(* IEC 61131-3 sources: YaoKangDeviceDemo/src/20_Decision, 3 files *)

(* ---- PRG_ErrorManager.st ---- *)
(*============================================================================
  PRG_ErrorManager —— 层 20 决策：错误与诊断（扫描链第 4 环），错误唯一写入者
  ----------------------------------------------------------------------------
  唯一写入：HMI.Sys.Error（当前活动错误）、HMI.Sys.Warning（警告通道）、
            HMI.Sys.ErrorQueue（9 条环形历史队列）；消费应答 gFaultSubmit:=FALSE。
  读入：  全局故障提交区 gFault*（各任务模块置位 gFaultSubmit 提交，本程序消费）；
          trigAckError / trigSysReset（错误确认/复位脉冲，由 INPUT_ADAPTER 锁存）；
          bSafetyStop（安全链态，活动 Critical 错误在安全链恢复前禁止清除）。
  提交约定：任务模块填 gFaultLevel/Code/Source/SubCode/Val1/Val2 后置
            gFaultSubmit:=TRUE；本程序入队并在同扫描清 gFaultSubmit。
            级别：0=L0 Info 1=L1 Warning 2=L2 Critical。
  清除语义：
    - Critical(L2) 进 Sys.Error 锁存，bNeedReset=TRUE，须 trigAckError/trigSysReset
      且安全链恢复(bSafetyStop=FALSE)才清除；复位不丢历史队列。
    - Warning(L1) 进 Sys.Warning，trigAckError 立即清除，否则存活 10s 自动消退。
    - 队列仅滚动追加，不随复位删除；bOverflow 记录溢出。
  说明：HMI.Sys.Display 的 iErrorCode/iErrorLevel/iErrorSubCode/iErrorSource 由
        HMI_OUTPUT 从 Sys.Error 镜像（单写源：Display 归 HMI_OUTPUT）。
        时间戳为毫秒运行刻度 diMsTick（上电起 ms，MONITOR 每扫累加 SCAN_PERIOD_MS）；
        非日历时钟，日志若需年月日时分秒待现场引入 RTC 库 FB 后替换（见 GVL_Internal diMsTick TODO）。
==========================================================================*)
PROGRAM PRG_ErrorManager

(*------------------------------------------------------------
  1) 故障消费：入队 + 活动错误/警告通道
------------------------------------------------------------*)
IF gFaultSubmit THEN
    (*--- 入环形队列：9 条，iTail 推进、iCount 计数、溢出置位 ---*)
    HMI.Sys.ErrorQueue.aEntries[HMI.Sys.ErrorQueue.iTail].iLevel      := gFaultLevel;
    HMI.Sys.ErrorQueue.aEntries[HMI.Sys.ErrorQueue.iTail].iCode       := gFaultCode;
    HMI.Sys.ErrorQueue.aEntries[HMI.Sys.ErrorQueue.iTail].iSource     := gFaultSource;
    HMI.Sys.ErrorQueue.aEntries[HMI.Sys.ErrorQueue.iTail].iVal1       := gFaultVal1;
    HMI.Sys.ErrorQueue.aEntries[HMI.Sys.ErrorQueue.iTail].diTimestamp := diMsTick;  (* 事件毫秒刻度（上电起 ms）；日历 RTC 待现场引入库 FB，见 GVL_Internal diMsTick TODO *)

    HMI.Sys.ErrorQueue.iTail := HMI.Sys.ErrorQueue.iTail + 1;
    IF HMI.Sys.ErrorQueue.iTail >= 9 THEN
        HMI.Sys.ErrorQueue.iTail := 0;
    END_IF;

    IF HMI.Sys.ErrorQueue.iCount < 9 THEN
        HMI.Sys.ErrorQueue.iCount := HMI.Sys.ErrorQueue.iCount + 1;
    ELSE
        HMI.Sys.ErrorQueue.iHead := HMI.Sys.ErrorQueue.iHead + 1;  (* 滚动覆盖最旧 *)
        IF HMI.Sys.ErrorQueue.iHead >= 9 THEN
            HMI.Sys.ErrorQueue.iHead := 0;
        END_IF;
        HMI.Sys.ErrorQueue.bOverflow := TRUE;
    END_IF;

    (*--- 当前活动错误 / 警告通道（L2→Error 锁存，L1→Warning 通道，L0 仅入队） ---*)
    IF gFaultLevel >= 2 THEN
        HMI.Sys.Error.iLevel     := gFaultLevel;
        HMI.Sys.Error.iCode      := gFaultCode;
        HMI.Sys.Error.iSource    := gFaultSource;
        HMI.Sys.Error.iSubCode   := gFaultSubCode;
        HMI.Sys.Error.iVal1      := gFaultVal1;
        HMI.Sys.Error.iVal2      := gFaultVal2;
        HMI.Sys.Error.bActive    := TRUE;
        HMI.Sys.Error.bCritical  := TRUE;
        HMI.Sys.Error.bEscalated := (gFaultCode = ERR_SOFT_ESTOP_TOUT);  (* 软急停超时升级硬急停 *)
        HMI.Sys.Error.bNeedReset := TRUE;    (* Critical 一律需手动复位 *)
    ELSIF gFaultLevel = 1 THEN
        HMI.Sys.Warning.iCode   := gFaultCode;
        HMI.Sys.Warning.iSource := gFaultSource;
        HMI.Sys.Warning.iVal1   := gFaultVal1;
        HMI.Sys.Warning.bActive := TRUE;
    END_IF;

    gFaultSubmit := FALSE;   (* 消费应答 *)
END_IF;

(*------------------------------------------------------------
  2) 活动 Critical 错误清除：确认/复位脉冲 + 安全链已恢复
     （安全链未恢复时拒绝清除，防止带故障复位运行）
------------------------------------------------------------*)
IF HMI.Sys.Error.bActive AND HMI.Sys.Error.bNeedReset THEN
    IF (trigAckError OR trigSysReset) AND NOT bSafetyStop THEN
        HMI.Sys.Error.bActive    := FALSE;
        HMI.Sys.Error.bCritical  := FALSE;
        HMI.Sys.Error.bEscalated := FALSE;
        HMI.Sys.Error.bNeedReset := FALSE;
        HMI.Sys.Error.iLevel     := 0;
        HMI.Sys.Error.iCode      := 0;
        HMI.Sys.Error.iSource    := 0;
        HMI.Sys.Error.iSubCode   := 0;
        HMI.Sys.Error.iVal1      := 0;
        HMI.Sys.Error.iVal2      := 0;
    END_IF;
END_IF;

(*------------------------------------------------------------
  3) 警告通道：确认即清；否则存活 10s 自动消退（实时态类警告）
------------------------------------------------------------*)
TONR(IN := HMI.Sys.Warning.bActive, PT := 10000, Q => emTWarnAge);  (* PT=DINT 毫秒：10s=10000ms *)
IF HMI.Sys.Warning.bActive THEN
    IF trigAckError OR emTWarnAge THEN
        HMI.Sys.Warning.bActive := FALSE;
        HMI.Sys.Warning.iCode   := 0;
        HMI.Sys.Warning.iSource := 0;
        HMI.Sys.Warning.iVal1   := 0;
    END_IF;
END_IF;

END_PROGRAM

(* ---- PRG_ModeManager.st ---- *)
(*============================================================================
  PRG_ModeManager —— 层 20 决策：系统状态机（扫描链第 6 环），iState 唯一写入者
  ----------------------------------------------------------------------------
  唯一写入：iState / iWorkMode / iUserRole / iBlockReason（全局）；
            Sys.Status 的 iState/iHealthLevel/diReadyCheckResult/bReady/
            bSafeToStart/bAutoProcessRunning/bIsEmergency/bNeedReset；
            离态残留电平命令（axisJogPos/axisJogNeg/jogPushUp/jogPushDown/pushEnableReq）。
  读入：  安全态 bHardEstop/bSoftEstop/bSafetyStop（最高优先级）；
          trig* 脉冲位（INPUT_ADAPTER 单扫锁存）、HMI.Sys.Cmd 的电平/INT 字段
          （iUserRole/iAuthCode/iWorkMode/bServiceAuthConfirm/bNoLoadConfirm）；
          资格位 bAllAxesIdle/Ref/AtInit、bParamBootDone/bRunParamValid；
          任务上报：Condition.Status.bDone/bError、HMI.Sys.Status.bSelfTestDone。
  规则：任务模块不直接切态，只上报 iPhase 与任务状态位；切换须过门控
        （角色/权限码/资格/安全），门控拒绝写 iBlockReason（45xx）供 HMI 提示；
        急停态无条件穿透；离态清残留电平命令。
  READY_CHECK：diReadyCheckResult 为位掩码（READY_MASK_*），0=全过；不齐时
        每 100 扫提交一次 7001 Warning，掩码值随 iVal1 上报。
==========================================================================*)
PROGRAM PRG_ModeManager

(*============================================================================
  0. 每扫公共计算：角色/工作模式镜像 + 六项资格掩码 + 汇总状态
  ==========================================================================*)
(*--- 工程师双重门控：角色 + 权限码 16#5A ---*)
mmBEngineer := (HMI.Sys.Cmd.iUserRole = ROLE_ENGINEER)
         AND (HMI.Sys.Cmd.iAuthCode = AUTH_CODE_ENGINEER);
iUserRole := HMI.Sys.Cmd.iUserRole;   (* 角色镜像（操作员/工程师） *)

(*--- 六项资格掩码（位值见 GVL_CONST READY_MASK_*，预计算位值直接 OR；LiteST 的 SHL/SHR 第一操作数不能是常量） ---*)
mmDiMask := 0;
IF NOT bAllAxesRef THEN
    mmDiMask := mmDiMask OR READY_MASK_REF;      (* bit5 参考无效 *)
END_IF;
IF NOT bRunParamValid OR NOT bParamBootDone THEN
    mmDiMask := mmDiMask OR READY_MASK_PARAM;   (* bit1 参数无效 *)
END_IF;
IF NOT HMI.Sys.Status.bPowerOn THEN
    mmDiMask := mmDiMask OR READY_MASK_HW;      (* bit2 硬件未上电 *)
END_IF;
IF HMI.Sys.Error.bActive THEN
    mmDiMask := mmDiMask OR READY_MASK_HEALTH;  (* bit3 活动 Critical *)
END_IF;
IF NOT bAllAxesAtInit THEN
    mmDiMask := mmDiMask OR READY_MASK_POS;     (* bit4 未在初始位 *)
END_IF;
IF NOT (retainZeroComm[0] AND retainZeroComm[1] AND retainZeroComm[2] AND retainTailZeroComm) THEN
    mmDiMask := mmDiMask OR READY_MASK_ZERO;    (* bit0 未建零 *)
END_IF;
mmBReadyAll := (mmDiMask = 0);

(*--- 汇总状态回填 Sys.Status ---*)
HMI.Sys.Status.iState             := iState;
HMI.Sys.Status.diReadyCheckResult := mmDiMask;
HMI.Sys.Status.bReady             := (iState = ST_STANDBY) AND mmBReadyAll;
HMI.Sys.Status.bSafeToStart       := mmBReadyAll AND (iState = ST_STANDBY)
                                AND NOT bSafetyStop AND NOT bHardEstop AND NOT bSoftEstop;
HMI.Sys.Status.bIsEmergency       := bHardEstop OR bSoftEstop OR bSafetyStop;
HMI.Sys.Status.bNeedReset         := HMI.Sys.Error.bNeedReset OR HMI.Sys.Error.bActive;
HMI.Sys.Status.bAutoProcessRunning:= (iState = ST_AUTORUN);
HMI.Sys.Status.iWorkMode          := iWorkMode;

(*--- 跳过自检资格位（P11） ---*)
(* 操作员快速启动：六项资格齐（含参考/建零），自检可安全省略；任何活动错误撤销资格 *)
HMI.Sys.Status.bSkipSelfTestAllowed := mmBReadyAll AND NOT HMI.Sys.Error.bActive;
(* 工程师强制跳过：需工程师双重门控（角色+权限码 16#5A），不受就绪位限制 *)
HMI.Sys.Status.bForceSkipSelfTestAllowed := mmBEngineer;

(*--- 健康等级 ---*)
IF HMI.Sys.Error.bActive THEN
    HMI.Sys.Status.iHealthLevel := HEALTH_FAULT;      (* 0 故障 *)
ELSIF HMI.Sys.Warning.bActive THEN
    HMI.Sys.Status.iHealthLevel := HEALTH_WARNING;    (* 2 警告 *)
ELSIF mmBReadyAll THEN
    HMI.Sys.Status.iHealthLevel := HEALTH_NORMAL;     (* 1 正常 *)
ELSE
    HMI.Sys.Status.iHealthLevel := HEALTH_UNKNOWN;    (* 3 未就绪 *)
END_IF;

(*--- 阻塞原因 iBlockReason（MODE_MANAGER 唯一写；稳态原因为主，下方 CASE 内
       工程师门控拒绝分支以 4503 覆盖本扫值）。安全/故障优先，其余按就绪缺项；
       0=无阻塞。与 diReadyCheckResult 掩码并行：掩码供调试，原因码供 HMI 显示。 ---*)
iBlockReason := 0;
IF bHardEstop OR bSoftEstop OR bSafetyStop THEN
    iBlockReason := BLOCK_REASON_SAFETY;   (* 4501 安全链动作（急停/保护停机中） *)
ELSIF HMI.Sys.Error.bActive THEN
    iBlockReason := BLOCK_REASON_FAULT;    (* 4502 活动 Critical，需复位 *)
ELSIF (iState = ST_STANDBY) OR (iState = ST_SERVICE_REQUIRED) THEN
    (* 待机/需服务为操作入口态：按就绪缺项给出最高优先原因（掩码细化见 diReadyCheckResult） *)
    IF NOT HMI.Sys.Status.bPowerOn THEN
        iBlockReason := BLOCK_REASON_POWER;      (* 4504 硬件未上电 *)
    ELSIF NOT (retainZeroComm[0] AND retainZeroComm[1] AND retainZeroComm[2] AND retainTailZeroComm) THEN
        iBlockReason := BLOCK_REASON_ZERO;       (* 4505 未建零，需维护建零 *)
    ELSIF NOT bRunParamValid OR NOT bParamBootDone THEN
        iBlockReason := BLOCK_REASON_PARAM;      (* 4506 运行参数无效 *)
    ELSIF NOT bAllAxesRef THEN
        iBlockReason := BLOCK_REASON_REF;        (* 4507 轴参考无效，需回零 *)
    ELSIF NOT bAllAxesAtInit THEN
        iBlockReason := BLOCK_REASON_POS;        (* 4508 未在初始位 *)
    END_IF;
END_IF;

(*============================================================================
  1. 急停最高优先级：任何状态无条件穿透
  ==========================================================================*)
IF bHardEstop THEN
    iState := ST_HARD_ESTOP;    (* 120 硬急停：断使能 *)
ELSIF bSoftEstop THEN
    iState := ST_SOFT_ESTOP;    (* 110 软急停：受控减速 *)
ELSE

    (* H5U：CASE 标签须用字面整数（具名常量按变量处理会报错），行尾注释码值 *)
    CASE iState OF

        (*---------- 0 上电初始化：参数首扫装载后转就绪检查 ----------*)
        0:
            IF bParamBootDone THEN
                iState := ST_READY_CHECK;    (* 3 *)
            END_IF;

        (*---------- 3 就绪检查：六项资格；齐→STANDBY，不齐节流报 7001 ----------*)
        3:
            IF trigReadyCheck OR mmBReadyAll THEN
                IF mmBReadyAll THEN
                    iState := ST_STANDBY;    (* 10 *)
                ELSE
                    mmIWarnDv := mmIWarnDv + 1;
                    IF mmIWarnDv >= 100 THEN
                        mmIWarnDv := 0;
                        gFaultLevel := 1;  gFaultCode := ERR_PRECHK_READY;
                        gFaultSource := SRC_MODE;  gFaultSubCode := 0;
                        gFaultVal1 := 0;  gFaultVal2 := 0;   (* 掩码见 Sys.Status.diReadyCheckResult *)
                        gFaultSubmit := TRUE;
                    END_IF;
                END_IF;
            END_IF;

        (*---------- 5 自检：任务完成→STANDBY；任务报错→STOPPING ----------*)
        5:
            IF trigSysStop THEN
                iState := ST_STOPPING;       (* 60 *)
            ELSIF HMI.Sys.Status.bSelfTestDone THEN
                iState := ST_STANDBY;        (* 10 *)
            END_IF;
            (* 自检失败由任务经 gFaultSubmit 提交 Critical，ErrorManager 置
               bNeedReset；本态检测到活动 Critical 即转 RESET 收口。 *)
            IF HMI.Sys.Error.bActive AND NOT HMI.Sys.Status.bSelfTestDone THEN
                iState := ST_RESET;          (* 50 *)
            END_IF;

        (*---------- 10 待机：全部门控入口 ----------*)
        10:
            (*--- 急停已在顶层穿透；停止/复位类 ---*)
            IF trigSysReset AND HMI.Sys.Error.bActive THEN
                iState := ST_RESET;          (* 50 *)
            (*--- 工程师门控拒绝：维护/标定/自检脉冲到但非工程师 → 4503（不切态） ---*)
            ELSIF (trigServiceMode OR trigCalibrate OR trigStartSelfTest) AND NOT mmBEngineer THEN
                iBlockReason := BLOCK_REASON_AUTH;   (* 4503 需工程师角色 + 权限码 16#5A *)
            (*--- 维护模式（工程师） ---*)
            ELSIF trigServiceMode AND mmBEngineer THEN
                iState := ST_SERVICE;        (* 30 *)
            (*--- 推杆标定（工程师） ---*)
            ELSIF trigCalibrate AND mmBEngineer THEN
                iState := ST_CALIBRATE;      (* 45 *)
            (*--- 回零（操作员/工程师均可；需硬件就绪） ---*)
            ELSIF trigSysHoming AND HMI.Sys.Status.bPowerOn THEN
                iState := ST_HOMING;         (* 40 *)
            (*--- 自检（工程师启动，或需强制跳过资格） ---*)
            ELSIF trigStartSelfTest AND mmBEngineer THEN
                iState := ST_SELFTEST;       (* 5 *)
            (*--- 自动流程：直接启动或快速启动（快速启动需资格位） ---*)
            ELSIF (trigAutoStart OR trigStart)
              AND (bSafeToStart OR (trigQuickStart AND HMI.Sys.Status.bSkipSelfTestAllowed)) THEN
                IF iWorkMode = 0 THEN
                    iWorkMode := HMI.Sys.Cmd.iWorkMode;   (* 锁存工作模式快照 *)
                END_IF;
                iState := ST_AUTORUN;        (* 20 *)
            END_IF;

        (*---------- 15 需要服务：仅工程师复位/维护可离开（保留态） ----------*)
        15:
            IF trigSysReset AND mmBEngineer THEN
                iState := ST_RESET;          (* 50 *)
            ELSIF trigServiceMode AND mmBEngineer THEN
                iState := ST_SERVICE;        (* 30 *)
            ELSIF (trigSysReset OR trigServiceMode) AND NOT mmBEngineer THEN
                iBlockReason := BLOCK_REASON_AUTH;   (* 4503 非工程师操作被拒 *)
            END_IF;

        (*---------- 20 自动流程运行：任务完成回 STANDBY；停止→STOPPING；急停顶层穿透 ----------*)
        20:
            IF trigSysStop OR trigStop THEN
                iState := ST_STOPPING;       (* 60 安全降落 *)
            ELSIF HMI.Condition.Status.bDone THEN
                iWorkMode := 0;
                iState := ST_STANDBY;        (* 10 完成 *)
            ELSIF HMI.Condition.Status.bEmergencyStop OR HMI.Condition.Status.bError THEN
                iState := ST_STOPPING;       (* 60 异常收口 *)
            END_IF;

        (*---------- 30 维护：维护完成回 STANDBY；可发起标定/回零（工程师） ----------*)
        30:
            IF trigServiceDone OR trigSysStop THEN
                iState := ST_STANDBY;        (* 10 *)
            ELSIF trigCalibrate THEN
                iState := ST_CALIBRATE;      (* 45 *)
            ELSIF trigSysHoming AND HMI.Sys.Status.bPowerOn THEN
                iState := ST_HOMING;         (* 40 *)
            END_IF;

        (*---------- 40 回零：回零完成→请求就绪检查；停止→STOPPING ----------*)
        40:
            IF trigSysStop THEN
                iState := ST_STOPPING;       (* 60 *)
            ELSIF bAllAxesRef AND bAllAxesAtInit AND bAllAxesIdle THEN
                (* 三轴参考有效且归初始位，维持 1s 稳定后由任务置 bHomeDone 收口；
                   此处仅以资格位判定完成，任务侧 iPhase=9 时回 STANDBY。 *)
                IF iPhase = COND_DONE THEN
                    iState := ST_STANDBY;    (* 10 *)
                END_IF;
            END_IF;
            IF HMI.Sys.Error.bActive THEN
                iState := ST_RESET;          (* 50 回零失败收口 *)
            END_IF;

        (*---------- 45 推杆标定：完成回原态（维护发起→SERVICE，待机发起→STANDBY） ----------*)
        45:
            IF trigSysStop THEN
                iState := ST_STOPPING;       (* 60 *)
            ELSIF HMI.TailTilt.Status.bCalibrated OR (iPhase = COND_DONE) THEN
                iState := ST_STANDBY;        (* 10（简化：标定完成回待机） *)
            END_IF;
            IF HMI.Sys.Error.bActive THEN
                iState := ST_RESET;          (* 50 标定失败收口 *)
            END_IF;

        (*---------- 50 复位收口：错误清除 + 轴复位后回 STANDBY ----------*)
        50:
            (* 复位任务（TaskRunner 50 分支）清 iPhase；待活动错误已被 ErrorManager
               清除且全轴静止，即回待机。残留 iState 写已从 TaskRunner 移除。 *)
            IF (NOT HMI.Sys.Error.bActive) AND bAllAxesIdle THEN
                iState := ST_STANDBY;        (* 10 *)
            END_IF;

        (*---------- 60 停止中：安全降落到初始位，停稳后回 STANDBY ----------*)
        60:
            IF bAllAxesIdle AND bAllAxesAtInit THEN
                iState := ST_STANDBY;        (* 10 *)
            END_IF;
            IF HMI.Sys.Error.bActive THEN
                iState := ST_RESET;          (* 50 停止中并发故障 *)
            END_IF;

        (*---------- 110 软急停：受控减速 + 紧急回零（任务）；解除+复位→RESET ----------*)
        110:
            IF (NOT bSafetyStop) AND trigSysReset THEN
                iState := ST_RESET;          (* 50 *)
            END_IF;

        (*---------- 120 硬急停：断使能；物理链恢复 + 复位→RESET ----------*)
        120:
            IF (NOT bSafetyStop) AND (NOT bHardEstopLatch) AND trigSysReset THEN
                iState := ST_RESET;          (* 50 *)
            END_IF;

        (*---------- 998 参数受限：保留（参数快照不一致等降级态），复位可回 STANDBY ----------*)
        998:

            IF trigSysReset AND mmBEngineer THEN
                iState := ST_RESET;          (* 50 *)
            ELSIF trigSysReset AND NOT mmBEngineer THEN
                iBlockReason := BLOCK_REASON_AUTH;   (* 4503 非工程师操作被拒 *)
            END_IF;

    ELSE
        iState := ST_INIT;    (* 0 未定义态兜底回上电 *)
    END_CASE;
END_IF;

(*============================================================================
  2. 离态清残留电平命令（安全约定）
     运动/点动类电平仅在明确许可的任务态有效；离开待机/维护进入自动/自检/
     回零/急停等态时，强制清零点动与推杆使能，防止跨态残留驱动。
     INPUT_ADAPTER 每扫先写电平位，本环在其后执行，故此处清零本扫生效。
     例外：软急停(ST_SOFT_ESTOP) 紧急回零 EMH_JOG_MAIN/CRAWL 需用三轴 Jog 电平
           受控回初始位（TaskRunner 环7 写 HMI.<Axis>.Cmd.bJogPos/Neg，InputAdapter
           环2 镜像 axisJogPos/Neg），故放行三轴点动；运动安全仍由 FB 内
           bSafetyStop 门控——软急停减速电平 smBSoftStopActive 未释放（轴未停稳）
           前 FB 不进 Jog 分支，EMH_WAIT_RELEASE 等其释放后才驱动。
           硬急停(ST_HARD_ESTOP) 不放行（断使能，点动无意义）。
           推杆点动任何急停态均清零（紧急回零不用推杆）。
  ==========================================================================*)
IF NOT ((iState = ST_STANDBY) OR (iState = ST_SERVICE) OR (iState = ST_SOFT_ESTOP)) THEN
    axisJogPos[0] := FALSE;  axisJogPos[1] := FALSE;  axisJogPos[2] := FALSE;
    axisJogNeg[0] := FALSE;  axisJogNeg[1] := FALSE;  axisJogNeg[2] := FALSE;
END_IF;
(* 推杆点动：非待机/维护一律清零（紧急回零不动作推杆） *)
IF NOT ((iState = ST_STANDBY) OR (iState = ST_SERVICE)) THEN
    jogPushUp   := FALSE;
    jogPushDown := FALSE;
END_IF;
(* 推杆使能仅在待机/维护/标定/回零/自动（成角段）允许；急停/复位/停止中断 *)
IF (iState = ST_HARD_ESTOP) OR (iState = ST_SOFT_ESTOP)
   OR (iState = ST_RESET) OR (iState = ST_STOPPING) THEN
    pushEnableReq := FALSE;
END_IF;

END_PROGRAM

(* ---- PRG_SafetyManager.st ---- *)
(*============================================================================
  PRG_SafetyManager —— 层 20 决策：安全防护（扫描链第 5 环），独立常驻
  ----------------------------------------------------------------------------
  唯一写入：bHardEstop / bSoftEstop / bProtStop / bHardEstopLatch / bSafetyStop；
            致命保护故障经 gFaultSubmit 提交（ERROR_MANAGER 入队）。
  读入：  ioEstopOK / ioEstop1 / ioEstop2（物理急停，去抖）；
          trigEmgStop（软急停脉冲）/ trigSysReset（复位脉冲，INPUT_ADAPTER 锁存，
          HMI 命令位已回清不可直读）；
          三轴 Status.Servo（bEncoderFault/bPosLimit/bNegLimit）、Force
          （bOverForce/bOverForceLatched）——OUTPUT_ADAPTER 镜像；
          推杆 Status.bError（堵转/超时由 FB_PusherControl 提交，本块不重复）。
  优先级：硬急停 > 软急停 > 保护停机；任何 iState 下都生效，不依赖业务状态。
  P4 落地：
    - 硬急停：物理链断开 OR 软急停超时升级锁存；断使能（POWER 读 bHardEstop）。
    - 双通道不一致诊断：两通道去抖态分歧持续 → 1003 Critical。
    - 软急停：HMI 脉冲锁存 bSoftEstop（事件/状态，驱动上报与 ModeManager 转 110），
      受控减速停车电平 smBSoftStopActive（驱动 bSafetyStop）；停稳持续 diEmergencyCoastMs
      后停车电平自动解除，放行 iState=110 紧急回零 Jog（bSoftEstop 仍保持，需
      trigSysReset 转 RESET）；减速 500 扫(≈5s)未全静止 → 升级锁存硬急停。
    - 保护停机：超力锁存 / 编码器故障（绝对位置不可信）→ bProtStop 受控减速锁存，
      需 trigSysReset 且条件消失才解除。
    - 硬限位（伺服 OriginSwitch 外的 bPosLimit/bNegLimit）→ 保护停机，脱限 Jog 由
      OUTPUT_ADAPTER 门控（不锁存，脱限即解除）。
    说明：扭矩防夹(1204)/推杆堵转(5001)/步骤超时由各运动 FB/任务就近提交。
==========================================================================*)
PROGRAM PRG_SafetyManager
VAR
    (* 上升沿：H5U 类型 TRIG.R_TRIG，仅局部 VAR 可声明，读 .Q。 *)
    rTrigHard      : TRIG.R_TRIG;
    rTrigSoft      : TRIG.R_TRIG;
    rTrigMismatch  : TRIG.R_TRIG;
    rTrigTimeout   : TRIG.R_TRIG;
    rTrigEncoder   : TRIG.R_TRIG;
    rTrigHwLimit   : TRIG.R_TRIG;
    rTrigOverForce : TRIG.R_TRIG;
    rTrigWatchdog  : TRIG.R_TRIG;
END_VAR

(*------------------------------------------------------------
  1) 诊断信号聚合（每扫合成；轴序 1=Chest 2=Seat 3=Leg）
------------------------------------------------------------*)
smBChanMismatch  := ioEstop1 <> ioEstop2;
smBAnyEncoderFlt := HMI.ChestImpact.Status.Servo.bEncoderFault
               OR HMI.SeatTwist.Status.Servo.bEncoderFault
               OR HMI.LegAngle.Status.Servo.bEncoderFault;
smBAnyHwLimit    := HMI.ChestImpact.Status.Servo.bPosLimit
               OR HMI.ChestImpact.Status.Servo.bNegLimit
               OR HMI.SeatTwist.Status.Servo.bPosLimit
               OR HMI.SeatTwist.Status.Servo.bNegLimit
               OR HMI.LegAngle.Status.Servo.bPosLimit
               OR HMI.LegAngle.Status.Servo.bNegLimit;
smBAnyOverForce  := HMI.ChestImpact.Status.Force.bOverForceLatched
               OR HMI.ChestImpact.Status.Force.bOverForce
               OR HMI.SeatTwist.Status.Force.bOverForceLatched
               OR HMI.SeatTwist.Status.Force.bOverForce
               OR HMI.LegAngle.Status.Force.bOverForceLatched
               OR HMI.LegAngle.Status.Force.bOverForce;

(*------------------------------------------------------------
  2) 急停链
------------------------------------------------------------*)
(* 2.1 双通道不一致：去抖 100ms 后判定（临界故障，拍急停安全侧，不单独驱动链） *)
TONR(IN := smBChanMismatch, PT := 100, Q => smTMismatch);  (* PT=DINT 毫秒：100ms *)

(* 2.2 软急停触发锁存：HMI 脉冲置位；trigSysReset（无硬急停/保护停机）解除。
       注意区分：bSoftEstop 是"发生过软急停"事件/状态锁存（驱动上报、ModeManager 转 110），
       smBSoftStopActive 是受控减速停车电平（驱动 bSafetyStop，使轴停止）。 *)
IF trigEmgStop AND NOT bHardEstop THEN
    bSoftEstop       := TRUE;
    smBSoftStopActive  := TRUE;   (* 停车电平同时置位 *)
ELSIF trigSysReset AND NOT (bHardEstop OR bProtStop) THEN
    bSoftEstop       := FALSE;
    smBSoftStopActive  := FALSE;
END_IF;

(* 2.3 软急停减速看门狗（500 扫 ≈ 5s）：停车电平有效但轴迟迟未全静止 → 升级锁存硬急停。
       计数仅在"减速中"（停车电平有效且未停稳）累加；停稳即清零（安全侧判据明确）。 *)
IF smBSoftStopActive AND NOT bAllAxesIdle AND NOT bHardEstopLatch THEN
    smDiSoftDecelCnt := smDiSoftDecelCnt + 1;
ELSE
    smDiSoftDecelCnt := 0;
END_IF;
IF smDiSoftDecelCnt >= 500 THEN
    bSoftEstop       := FALSE;   (* 软急停升级为硬急停，软态让位 *)
    smBSoftStopActive  := FALSE;
    bHardEstopLatch  := TRUE;
END_IF;

(* 2.3b 紧急回零放行（设计点①）：软急停受控减速停稳（bAllAxesIdle 持续
       diEmergencyCoastMs，默认 500ms=50 扫）后，自动解除减速停车电平，
       使 TASK_RUNNER 在 iState=110 内可发受控 Jog 回初始位。系统仍处软急停状态
       （bSoftEstop 保持，ModeManager 仍需 trigSysReset 转 RESET）；防夹由任务层
       rNetTorquePct 超阈兜底。再发 trigEmgStop 重新置位停车电平（立即二次减速）。 *)
IF smBSoftStopActive AND bAllAxesIdle THEN
    smDiCoastCnt := smDiCoastCnt + 1;
ELSE
    smDiCoastCnt := 0;
END_IF;
IF smBSoftStopActive AND (smDiCoastCnt >= runHoming.diEmergencyCoastMs / 10) THEN
    smBSoftStopActive := FALSE;   (* 停车电平解除，允许紧急 Jog；bSoftEstop 状态仍保持 *)
    smDiCoastCnt      := 0;
END_IF;

(* 2.4 硬急停：物理链断开（瞬时）OR 超时升级锁存。
       锁存解除：物理链恢复 + 复位脉冲（物理急停未恢复前禁止解除）。 *)
bHardEstop := (NOT ioEstopOK) OR bHardEstopLatch;
IF bHardEstopLatch AND ioEstopOK AND trigSysReset THEN
    bHardEstopLatch := FALSE;
END_IF;

(*------------------------------------------------------------
  3) 保护停机（受控减速后锁死，区别于硬急停断使能）
------------------------------------------------------------*)
(* 3.1 超力锁存：牵引力超阈持续（Force.bOverForceLatched 由 OUTPUT_ADAPTER 置位） *)
IF smBAnyOverForce THEN
    bProtStop := TRUE;
END_IF;
(* 3.2 编码器故障：绝对位置不可信，禁定位类动作，立即受控停机 *)
IF smBAnyEncoderFlt THEN
    bProtStop := TRUE;
END_IF;
(* 3.3 解除：复位脉冲 + 全部触发条件消失 *)
IF bProtStop AND trigSysReset AND NOT smBAnyOverForce AND NOT smBAnyEncoderFlt THEN
    bProtStop := FALSE;
END_IF;

(* 硬限位不锁存：OUTPUT_ADAPTER 禁越限运动并提供脱限 Jog；脱限即自然解除。
   软限位(2004 警告)由运动 FB 判定提交，不在此驱动停机。 *)

(*------------------------------------------------------------
  4) 安全停止合成（POWER 断使能判 bHardEstop；OUTPUT_ADAPTER 减速判 bSafetyStop）
------------------------------------------------------------*)
bSafetyStop := bHardEstop OR smBSoftStopActive OR bProtStop OR smBAnyHwLimit;

(*------------------------------------------------------------
  5) 事件上报（上升沿提交一次；每扫至多一条，优先级按安全严重度）
------------------------------------------------------------*)
smBHardPhysical := NOT ioEstopOK;     (* 物理链断开（不含锁存升级） *)
rTrigHard(CLK     := smBHardPhysical);
rTrigMismatch(CLK := smTMismatch);
rTrigTimeout(CLK  := bHardEstopLatch);
rTrigSoft(CLK     := bSoftEstop);
rTrigEncoder(CLK  := smBAnyEncoderFlt);
rTrigHwLimit(CLK  := smBAnyHwLimit);
rTrigOverForce(CLK := smBAnyOverForce);
rTrigWatchdog(CLK := mnTScanWatchdog);

(* 扫描看门狗 1007：本位预留，正常不置位（真实看门狗为 H5U 任务组态/硬件，
   超时由控制器停机/进安全态；详见 PRG_Main 注释）。一旦被系统变量置位，
   作为最高优先级 Critical 上报一次，交 ModeManager 转 RESET 收口。处置策略待现场确认。 *)
IF rTrigWatchdog.Q THEN
    gFaultLevel := 2; gFaultCode := ERR_SCAN_WATCHDOG; gFaultSource := SRC_SAFETY;
    gFaultSubCode := 0; gFaultVal1 := 0; gFaultVal2 := 0;
    gFaultSubmit := TRUE;
ELSIF rTrigHard.Q THEN
    gFaultLevel := 2; gFaultCode := ERR_HARD_ESTOP; gFaultSource := SRC_SAFETY;
    gFaultSubCode := 0; gFaultVal1 := 0; gFaultVal2 := 0;
    gFaultSubmit := TRUE;
ELSIF smTMismatch AND rTrigMismatch.Q THEN
    gFaultLevel := 2; gFaultCode := ERR_ESTOP_MISMATCH; gFaultSource := SRC_SAFETY;
    gFaultSubCode := 0; gFaultVal1 := BOOL_TO_INT(ioEstop1); gFaultVal2 := BOOL_TO_INT(ioEstop2);
    gFaultSubmit := TRUE;
ELSIF rTrigTimeout.Q THEN
    gFaultLevel := 2; gFaultCode := ERR_SOFT_ESTOP_TOUT; gFaultSource := SRC_SAFETY;
    gFaultSubCode := 0; gFaultVal1 := 0; gFaultVal2 := 0;
    gFaultSubmit := TRUE;
ELSIF rTrigSoft.Q THEN
    gFaultLevel := 2; gFaultCode := ERR_SOFT_ESTOP; gFaultSource := SRC_SAFETY;
    gFaultSubCode := 0; gFaultVal1 := 0; gFaultVal2 := 0;
    gFaultSubmit := TRUE;
ELSIF rTrigOverForce.Q THEN
    gFaultLevel := 2; gFaultCode := ERR_OVERFORCE; gFaultSource := SRC_SAFETY;
    gFaultSubCode := 0; gFaultVal1 := 0; gFaultVal2 := 0;
    gFaultSubmit := TRUE;
ELSIF rTrigEncoder.Q THEN
    gFaultLevel := 2; gFaultCode := ERR_AXIS_ENCODER; gFaultSource := SRC_SAFETY;
    gFaultSubCode := 0; gFaultVal1 := BOOL_TO_INT(smBAnyEncoderFlt); gFaultVal2 := 0;
    gFaultSubmit := TRUE;
ELSIF rTrigHwLimit.Q THEN
    gFaultLevel := 2; gFaultCode := ERR_AXIS_HWLIMIT; gFaultSource := SRC_SAFETY;
    gFaultSubCode := 0; gFaultVal1 := 0; gFaultVal2 := 0;
    gFaultSubmit := TRUE;
END_IF;

END_PROGRAM
